VISUALIZATION _VISU_PcMiniVertical  // 10x120
VAR_IN_OUT
  m_Inst  : FB_PC;
END_VAR
    RoundedRectangle (0,0 10x100), colour toggle: m_Inst._bBoardEnable
    RoundedRectangle (0,50 10x10), "J", tooltip "Job loaded", colour toggle: NOT m_Inst._sPcFlags.bQueueEmpty AND NOT m_Inst._sPcFlags.bError
    RoundedRectangle (0,60 10x10), "I", colour toggle: m_Inst._sPcState.bIdle
    RoundedRectangle (0,70 10x10), "R", colour toggle: m_Inst._sPcState.bReady
    RoundedRectangle (0,80 10x10), "P", colour toggle: m_Inst._sPcState.bPrinting
    RoundedRectangle (0,90 10x10), "D", colour toggle: m_Inst._sPcState.bDone
    RoundedRectangle (0,110 10x10), "C", tooltip "Communication error", colour toggle: m_Inst.sI_PhHw.ecWcState, invisible if: NOT m_Inst.sI_PhHw.ecWcState
    RoundedRectangle (0,100 10x10), "E", tooltip "Error", invisible if: NOT m_Inst._sPcFlags.bError
    RoundedRectangle (0,0 10x100), "E"
        toggle m_Inst._pAds^.bI_Enable
    Ellipse (0,30 10x10), tooltip "Heater enable"
        toggle PRG_PRINT.sAdsPrintController[1].sI_EnableHeater.bI_SetBool
    Ellipse (0,40 10x10), tooltip "Print enable"
        toggle PRG_PRINT.sAdsPrintController[1].sI_EnablePrint.bI_SetBool
END_VISUALIZATION

(* stored: Version 1.1.0.1, ProductVersion 3.1.4024.11
   Visu _VISU_PcMiniVertical: Id {8c35e159-baf9-4292-8da6-479cd8b48198} *)
